// TIA Portal V20 export
DATA_BLOCK "Config"   // DB153
// stored: MemoryReserve 100, Namespace Unit1.Em0
   VAR
      em : "LAF_typeEmConfiguration";   // Configuration of EM Parameters
      axis : Array[1.._.U1EM0_NO_OF_AXES] of DB_ANY;
      moduleAccessPoint : Array[1.._.U1EM0_NO_OF_AXES] of HW_SUBMODULE;
   END_VAR
   VAR RETAIN
      cmUnWinderAxisB : "LBC_typeAxisControlConfiguration";
      cmAirShaftOnOff : "LBC_typeTwoWayActuatorConfiguration";
      cmExpelFwdBwd : "LBC_typeTwoWayActuatorConfiguration";
      cmTensionCheckSensor : "LBC_typeDigitalSignalConfiguration";
      cmRadiusMeasureAnalogInput : "LBC_typeAnalogInputConfiguration";
      cmEpc : "LER_typeCON600Configuration";
      cmRadiusMeasure : "LER_typeRadiusMeasureConfiguration";
      cmUnWinderAxisB_TorqueCal : "LER_typeServoTorqueCalConfigruation";
   END_VAR
BEGIN
   // axis[1] : cmUnWinderAxisB
   // moduleAccessPoint[1] : cmUnWinderAxisB
END_DATA_BLOCK
